// TIA Portal V17 export
BLOCK "FC_CallEno"   // ObjectSW17, LAD
BEGIN

REGION Network 1: call with eno
END_REGION
END_BLOCK
